FUNCTION_BLOCK PIDBase (* Composite Function Block Type *)
  (* Standard: 61499-2 *)
  (* Version 1.0.1, 10/18/2023, ApplicationLibDevTeam, Schneider Electric, First Version *)
  PACKAGE Main;
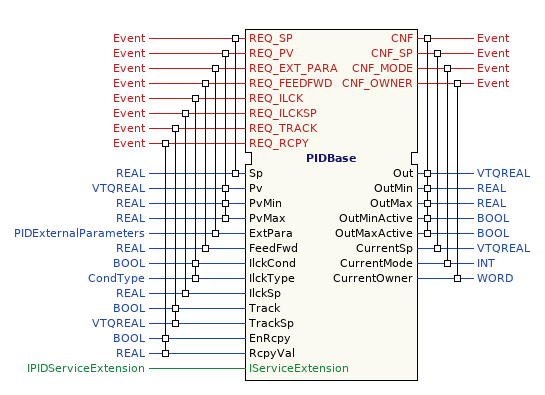
  EVENT_INPUT
    REQ_SP WITH Sp; (* Request to update setpoint *)
    REQ_PV WITH Pv, PvMin, PvMax; (* Request to update input value *)
    REQ_EXT_PARA WITH ExtPara; (* Request to update external PID parameters *)
    REQ_FEEDFWD WITH FeedFwd; (* Request for executing feed forward gain *)
    REQ_ILCK WITH IlckCond, IlckType; (* Request to update interlock conditions *)
    REQ_ILCKSP WITH IlckSp; (* Request to update interlock setpoint to PID ouput *)
    REQ_TRACK WITH Track, TrackSp; (* Request to track PID setpoint with TrackState *)
    REQ_RCPY WITH EnRcpy, RcpyVal; (* Request for actuator position *)
  END_EVENT
  EVENT_OUTPUT
    CNF WITH Out, OutMinActive, OutMaxActive, OutMin, OutMax; (* Execution confirmation (Cyclic update) *)
    CNF_SP WITH CurrentSp; (* Execution confirmation of current setpoint *)
    CNF_MODE WITH CurrentMode; (* Execution of confirmation of current mode *)
    CNF_OWNER WITH CurrentOwner; (* Execution confirmation of owner *)
  END_EVENT
  VAR_INPUT
    Sp : REAL; (* Setpoint for PID calculation *)
    Pv : VTQREAL; (* Unscaled analog process value *)
    PvMin : REAL; (* Minimum range of process value *)
    PvMax : REAL; (* Maximum range of process value *)
    ExtPara : PIDExternalParameters; (* External parameters for PID calculation *)
    FeedFwd : REAL; (* Feed forward value *)
    IlckCond : BOOL; (* 1 = Interlock condition active *)
    IlckType : CondType; (* Type of condition interlock, (0 = Normal, 1 = Process interlock/Sequence interlock) *)
    IlckSp : REAL; (* Interlock setpoint *)
    Track : BOOL; (* 1 = Track calclated output to TrackSp *)
    TrackSp : VTQREAL; (* If Track enabled, PID ouput follows TrackSp (Out = TrackSp) *)
    EnRcpy : BOOL; (* 1 = the RCPY is enabled *)
    RcpyVal : REAL; (* RCPY value (actuator position) *)
  END_VAR
  VAR_OUTPUT
    Out : VTQREAL; (* Calculated output value *)
    OutMin : REAL; (* Minimum range of ouput value *)
    OutMax : REAL; (* Maximum range of ouput value *)
    OutMinActive : BOOL; (* 1 = Out has reached OutMin Limit *)
    OutMaxActive : BOOL; (* 1 = Out has reached OutMax Limit *)
    CurrentSp : VTQREAL; (* Current setpoint value *)
    CurrentMode : INT; (* Current mode selected for PID calculation *)
    CurrentOwner : WORD; (* Current owner data from externlal source and basic owner 16#8 = Program owner, 16#10 = Operator owner, 16#4 = program Local and 16#40 Operator Local *)
  END_VAR
  SOCKETS
    IServiceExtension : IPIDServiceExtension(ServiceState := TRUE); (* Services extension adapter(Seq control and Owner) *)
  END_SOCKETS
  (* Initialization *)
  (* Supervision Interface *)
  (* Control *)
  (* Owner & Setpoint Management *)
  (* Data exchange with sequence *)
  (* Parameter Selection *)
  FBS
    IThis : PIDBase_HMI(QI := TRUE);
    plcStart : plcStart(Delay := T#0ms, Prio := 16);
    setpointRamp : rampCtl(MaxDeviation := 0.0, EnableDeviation := FALSE);
    pidCalc : pidCtl(ProhibitOutInc := FALSE, ProhibitOutDec := FALSE);
    modeSelection : devInSel(EnBumpless1 := FALSE, Val1 := (value:=0,quality:=16#0,timestamp:=LDT#2023-10-14-17:35:08,picosecs:=0), EnBumpless2 := TRUE, EnBumpless3 := FALSE, PermPassive := FALSE, PermActive1 := FALSE, PermActive2 := FALSE, UseCurrentVal := TRUE); {SET_ATTRIBUTE(Configuration.Component.HideUnusedPorts, )}
    basicOwner : ownerControl;
    programModeSelection : SELECT_24363B89CFDE21263(IN1 := 1); {SET_ATTRIBUTE(Configuration.GenericFBType.InterfaceParams, Runtime.Standard#CNT:=2;SELECT:BOOL;IN${CNT$}:INT)}
    spSelection : devRealSel(EnBumpless2 := TRUE, EnBumpless3 := FALSE, EnBumpless1 := FALSE); {SET_ATTRIBUTE(Configuration.Component.HideUnusedPorts, )}
    programSpSelection : SELECT_218F0E76F8A148ECD; {SET_ATTRIBUTE(Configuration.GenericFBType.InterfaceParams, Runtime.Standard#CNT:=2;SELECT:BOOL;IN${CNT$}:REAL)}
    outSelection : devRealSel(EnBumpless2 := FALSE, EnBumpless3 := TRUE, EnBumpless1 := FALSE, EnBumpless4 := FALSE, EnBumpless5 := FALSE); {SET_ATTRIBUTE(Configuration.Component.HideUnusedPorts, )}
    modeCalc : modeCalc;
    trackingActive : E_SELECT;
    paraSel : DS_SELECTX_125F0E43806CD1F46; {SET_ATTRIBUTE(Configuration.GenericFBType.InterfaceParams, Runtime.Standard#CNTX:=2;CNTY:=9;DI${CNTX,_,CNTY$}:REAL,REAL,REAL,BOOL,REAL,BOOL,REAL,REAL,REAL)} {SET_ATTRIBUTE(Configuration.Component.HideUnusedPorts, )}
    extParaSel : E_SWITCH;
    paraSelectionCheck : DS_SELECTX_4480AAC7B40EACCE; {SET_ATTRIBUTE(Configuration.GenericFBType.InterfaceParams, Runtime.Standard#CNTX:=2;CNTY:=10;DI${CNTX,_,CNTY$}:BOOL,REAL,REAL,REAL,BOOL,REAL,BOOL,REAL,REAL,REAL)}
    extParaCheck : E_SWITCH;
    paraSplit : SPLIT_62F891E498C2EEC3; {SET_ATTRIBUTE(Configuration.GenericFBType.InterfaceParams, Runtime.Standard#<InterfaceList> <EventInputs> <Event Name="REQ" Comment="Request events for dedicated input data sets"> <With Var="Input" /> </Event> </EventInputs> <EventOutputs> <Event Name="CNF" Comment="Confirmation from Resource for a dedicated request"> <With Var="Output" /> <With Var="Enable" /> <With Var="Gain" /> <With Var="IntegralTime" /> <With Var="DerivationTime" /> <With Var="Directon" /> <With Var="DeadBand" /> <With Var="DWorkOnError" /> <With Var="LagTime" /> <With Var="OutMin" /> <With Var="OutMax" /> </Event> </EventOutputs> <InputVars> <VarDeclaration Name="Input" Type="PIDExternalParameters" Namespace="SE.App2CommonProcess" /> </InputVars> <OutputVars> <VarDeclaration Name="Output" Type="PIDExternalParameters" Namespace="SE.App2CommonProcess" /> <VarDeclaration Name="Enable" Type="BOOL" /> <VarDeclaration Name="Gain" Type="REAL" /> <VarDeclaration Name="IntegralTime" Type="REAL" /> <VarDeclaration Name="DerivationTime" Type="REAL" /> <VarDeclaration Name="Directon" Type="BOOL" /> <VarDeclaration Name="DeadBand" Type="REAL" /> <VarDeclaration Name="DWorkOnError" Type="BOOL" /> <VarDeclaration Name="LagTime" Type="REAL" /> <VarDeclaration Name="OutMin" Type="REAL" /> <VarDeclaration Name="OutMax" Type="REAL" /> </OutputVars> </InterfaceList>)}
  END_FBS
  EVENT_CONNECTIONS
    modeSelection.CNF TO CNF_MODE;
    programSpSelection.CNF TO spSelection.REQ_SP3;
    programModeSelection.CNF TO modeSelection.REQ_SP3;
    IServiceExtension.REQ_OWNER TO basicOwner.REQ_STDOWNER;
    spSelection.CNF TO CNF_SP;
    REQ_TRACK TO modeSelection.REQ_SP1;
    REQ_ILCK TO outSelection.REQ_SEL;
    REQ_TRACK TO modeCalc.REQ_TRACK;
    REQ_TRACK TO outSelection.REQ_SP1;
    modeCalc.CNF TO outSelection.REQ_SEL;
    modeCalc.CNF_TRACK TO outSelection.REQ_SEL;
    REQ_ILCKSP TO outSelection.REQ_SP2;
    pidCalc.C_CNF TO outSelection.REQ_SP5;
    outSelection.CNF TO pidCalc.REQ;
    modeSelection.CNF TO modeCalc.REQ_MODE;
    modeCalc.CNF_TRACK TO modeSelection.REQ_SEL;
    IServiceExtension.REQ_CMD TO programModeSelection.REQ;
    IServiceExtension.REQ_SP TO programSpSelection.REQ;
    REQ_SP TO programSpSelection.REQ;
    REQ_PV TO pidCalc.REQ;
    modeCalc.CNF TO spSelection.REQ_SEL;
    REQ_PV TO spSelection.REQ_SP1;
    modeCalc.CNF TO setpointRamp.REQ_TRACK;
    spSelection.CNF TO setpointRamp.REQ_SP;
    modeSelection.CNF TO IServiceExtension.CNF_MODE;
    REQ_PV TO setpointRamp.REQ_SP;
    setpointRamp.CNF TO pidCalc.REQ_SP;
    REQ_FEEDFWD TO pidCalc.REQ_FEEDFWD;
    modeCalc.CNF_MODE TO pidCalc.REQ;
    REQ_PV TO setpointRamp.REQ_TRACK;
    REQ_ILCK TO IServiceExtension.CNF_READY;
    REQ_PV TO IServiceExtension.CNF_PV;
    setpointRamp.CNF TO IServiceExtension.CNF_SP_OP;
    plcStart.FIRST_INIT TO IServiceExtension.CNF_SERVICE;
    pidCalc.CNF_READY TO IServiceExtension.CNF_READY;
    basicOwner.CNF_OWNER TO modeCalc.REQ_OWNER;
    pidCalc.C_CNF TO trackingActive.EI0;
    trackingActive.EO TO CNF;
    modeCalc.CNF_TRACK TO trackingActive.EI0;
    trackingActive.EO TO IServiceExtension.CNF_SP_OP;
    pidCalc.CNF TO trackingActive.EI1;
    extParaSel.EO1 TO paraSel.REQ2;
    paraSel.IND TO pidCalc.REQ_PARA;
    REQ_TRACK TO pidCalc.REQ_TRACK;
    IServiceExtension.REQ_PARA TO extParaCheck.EI;
    extParaCheck.EO0 TO paraSelectionCheck.REQ1;
    extParaCheck.EO1 TO paraSelectionCheck.REQ2;
    REQ_EXT_PARA TO paraSplit.REQ;
    paraSplit.CNF TO extParaCheck.EI;
    IServiceExtension.REQ_OUT TO outSelection.REQ_SP4;
    REQ_ILCK TO modeCalc.REQ_ILCK;
    basicOwner.CNF_OWNER TO programModeSelection.REQ;
    REQ_TRACK TO IServiceExtension.CNF_TRACK;
    REQ_ILCK TO pidCalc.REQ_ILCK;
    modeCalc.CNF TO modeSelection.REQ_SEL;
    basicOwner.CNF_OWNER TO CNF_OWNER;
    paraSel.IND TO IServiceExtension.CNF_SP_OP;
    paraSel.IND TO IServiceExtension.8CDB19EE4FC593B1;
    paraSelectionCheck.IND TO extParaSel.EI;
    plcStart.FIRST_INIT TO IThis.F4ED48CC2B5317F8;
    IThis.3C7816C1E3C12126 TO IThis.F8BDFB66D6A721B;
    modeCalc.CNF TO IThis.4ECF71528D4B6340;
    REQ_ILCK TO IThis.4ECF71528D4B6340;
    REQ_PV TO IThis.4ECF71528D4B6340;
    setpointRamp.CNF TO IThis.4ECF71528D4B6340;
    pidCalc.CNF TO IThis.4ECF71528D4B6340;
    modeCalc.CNF_MODE TO IThis.4ECF71528D4B6340;
    REQ_TRACK TO IThis.4ECF71528D4B6340;
    pidCalc.C_CNF TO IThis.4ECF71528D4B6340;
    spSelection.CNF TO IThis.4ECF71528D4B6340;
    modeCalc.CNF_TRACK TO IThis.568B5274285BDEC8;
    paraSel.IND TO IThis.568B5274285BDEC8;
    extParaSel.EO0 TO IThis.568B5274285BDEC8;
    IThis.3C7816C1E3C12126 TO basicOwner.REQ_BASICOWNER;
    IThis.3C7816C1E3C12126 TO plcStart.ACK_FIRST;
    IThis.CF580EC7DC4C111C TO basicOwner.REQ_BASICOWNER;
    IThis.733DF8FD825824CA TO spSelection.REQ_SP2;
    IThis.F7A34A5B968DDB98 TO outSelection.REQ_SP3;
    IThis.DF1716734AF61076 TO setpointRamp.REQ_PARA;
    IThis.DF1716734AF61076 TO modeCalc.REQ_OWNER;
    IThis.DF1716734AF61076 TO paraSel.REQ1;
    IThis.D88CEB590B668985 TO modeSelection.REQ_SP2;
    IThis.D88CEB590B668985 TO setpointRamp.REQ_PARA;
    IThis.D88CEB590B668985 TO paraSel.REQ1;
    IThis.D716EC33D901A5A4 TO pidCalc.REQ_OUTBIAS;
    REQ_RCPY TO pidCalc.F3BAF1D546068DF6;
  END_CONNECTIONS
  DATA_CONNECTIONS
    modeSelection.CurrentVal TO CurrentMode;
    Sp TO programSpSelection.IN1;
    programSpSelection.OUT TO spSelection.Val3;
    programModeSelection.OUT TO modeSelection.Val3;
    basicOwner.ProgramOwner TO modeSelection.Sel3;
    basicOwner.OperatorOwner TO modeSelection.Sel2;
    basicOwner.StdOwnerConnected TO programModeSelection.SELECT;
    basicOwner.ProgramOwner TO spSelection.Sel3;
    basicOwner.StdOwnerConnected TO programSpSelection.SELECT;
    IServiceExtension.StdOwner TO basicOwner.StdOwner;
    spSelection.CurrentVal TO CurrentSp;
    TrackSp TO outSelection.Val1;
    Track TO modeSelection.Sel1;
    IlckSp TO outSelection.Val2;
    IlckCond TO outSelection.Sel2;
    Track TO outSelection.Sel1;
    Track TO modeCalc.Track;
    modeSelection.CurrentVal TO modeCalc.ModeIn;
    pidCalc.Out TO outSelection.Val5;
    outSelection.CurrentVal TO pidCalc.PresetValue;
    modeCalc.ModeOut TO outSelection.Sel5;
    modeCalc.OperManual TO outSelection.Sel3;
    IServiceExtension.Sp TO programModeSelection.IN2;
    IServiceExtension.SpReal1 TO programSpSelection.IN2;
    modeCalc.TrackManual TO spSelection.Sel1;
    Pv TO pidCalc.Pv;
    Pv TO spSelection.Val1;
    modeCalc.TrackManual TO setpointRamp.Track;
    IlckCond TO modeCalc.IlckCond;
    spSelection.CurrentVal TO setpointRamp.Sp;
    modeSelection.CurrentVal TO IServiceExtension.CurrentMode;
    PvMin TO setpointRamp.SpMin;
    PvMax TO setpointRamp.SpMax;
    Pv TO setpointRamp.TrackSp;
    setpointRamp.Out TO pidCalc.Sp;
    FeedFwd TO pidCalc.FeedFwd;
    IlckCond TO IServiceExtension.Interlocked;
    pidCalc.Out TO IServiceExtension.CurrentOp;
    setpointRamp.Out TO IServiceExtension.CurrentSp;
    Pv TO IServiceExtension.Pv;
    pidCalc.Out TO Out;
    pidCalc.OutMinActive TO OutMinActive;
    pidCalc.OutMaxActive TO OutMaxActive;
    IlckType TO pidCalc.IlckType;
    IlckCond TO pidCalc.IlckCond;
    pidCalc.Ready TO IServiceExtension.Ready;
    Track TO pidCalc.TrackSp;
    modeCalc.OperAuto TO spSelection.Sel2;
    basicOwner.Owner TO modeCalc.Owner;
    Track TO trackingActive.G;
    modeCalc.ProgLocalManual TO outSelection.Sel4;
    paraSel.OUT1 TO pidCalc.Gain;
    paraSel.OUT2 TO pidCalc.IntegralTime;
    paraSel.OUT3 TO pidCalc.DerivativeTime;
    paraSel.OUT4 TO pidCalc.Direction;
    paraSel.OUT5 TO pidCalc.Deadband;
    paraSel.OUT6 TO pidCalc.DWorkOnError;
    paraSel.OUT7 TO pidCalc.LagTime;
    paraSel.OUT8 TO pidCalc.OutMin;
    paraSel.OUT9 TO pidCalc.OutMax;
    IServiceExtension.ExtParaSel TO extParaCheck.G;
    IServiceExtension.Gain TO paraSelectionCheck.DI2_2;
    IServiceExtension.IntegralTime TO paraSelectionCheck.DI2_3;
    IServiceExtension.DerivationTime TO paraSelectionCheck.DI2_4;
    IServiceExtension.Direction TO paraSelectionCheck.DI2_5;
    IServiceExtension.DeadBand TO paraSelectionCheck.DI2_6;
    IServiceExtension.DWorkOnError TO paraSelectionCheck.DI2_7;
    IServiceExtension.LagTime TO paraSelectionCheck.DI2_8;
    IServiceExtension.OutMin TO paraSelectionCheck.DI2_9;
    IServiceExtension.OutMax TO paraSelectionCheck.DI2_10;
    paraSel.OUT8 TO OutMin;
    paraSel.OUT9 TO OutMax;
    paraSelectionCheck.OUT10 TO paraSel.DI2_9;
    paraSelectionCheck.OUT2 TO paraSel.DI2_1;
    paraSelectionCheck.OUT3 TO paraSel.DI2_2;
    paraSelectionCheck.OUT4 TO paraSel.DI2_3;
    paraSelectionCheck.OUT5 TO paraSel.DI2_4;
    paraSelectionCheck.OUT6 TO paraSel.DI2_5;
    paraSelectionCheck.OUT7 TO paraSel.DI2_6;
    paraSelectionCheck.OUT8 TO paraSel.DI2_7;
    paraSelectionCheck.OUT9 TO paraSel.DI2_8;
    IServiceExtension.ExtParaSel TO paraSelectionCheck.DI2_1;
    paraSelectionCheck.OUT1 TO extParaSel.G;
    ExtPara TO paraSplit.Input;
    paraSplit.Enable TO paraSelectionCheck.DI1_1;
    paraSplit.Gain TO paraSelectionCheck.DI1_2;
    paraSplit.IntegralTime TO paraSelectionCheck.DI1_3;
    paraSplit.DerivationTime TO paraSelectionCheck.DI1_4;
    paraSplit.Directon TO paraSelectionCheck.DI1_5;
    paraSplit.DeadBand TO paraSelectionCheck.DI1_6;
    paraSplit.DWorkOnError TO paraSelectionCheck.DI1_7;
    paraSplit.LagTime TO paraSelectionCheck.DI1_8;
    paraSplit.OutMin TO paraSelectionCheck.DI1_9;
    paraSplit.OutMax TO paraSelectionCheck.DI1_10;
    IServiceExtension.SpReal2 TO outSelection.Val4;
    modeCalc.CalcMode TO pidCalc.Mode;
    Track TO IServiceExtension.Track;
    basicOwner.Owner TO CurrentOwner;
    PvMin TO IServiceExtension.PvMin;
    PvMax TO IServiceExtension.PvMax;
    paraSel.OUT8 TO IServiceExtension.CurrentOpMin;
    paraSel.OUT9 TO IServiceExtension.CurrentOpMax;
    paraSel.OUT1 TO IServiceExtension.526988CF984C619A;
    paraSel.OUT2 TO IServiceExtension.7D8F5388E2DC486D;
    paraSel.OUT3 TO IServiceExtension.B62ECEA2F5E6DA8A;
    paraSel.OUT4 TO IServiceExtension.607F2E8B0E693249;
    paraSel.OUT5 TO IServiceExtension.60EB9615BA837102;
    paraSel.OUT6 TO IServiceExtension.3F4910500F1CC6A6;
    paraSel.OUT7 TO IServiceExtension.B38B3033E4F94F3F;
    Pv TO IThis.ACDC6904590859A8;
    PvMin TO IThis.8881FFD24D90D865;
    PvMax TO IThis.E15A9214DEEE85B6;
    spSelection.CurrentVal TO IThis.AA9BE811C6AB052A;
    pidCalc.Out TO IThis.F680A73B417CD6F5;
    modeSelection.CurrentVal TO IThis.5BB4B57D9CC10C19;
    basicOwner.Owner TO IThis.3143D32BCC6D529B;
    pidCalc.OutChangeProhibited TO IThis.38051CE7590A4498;
    Track TO IThis.F23EE025A922C157;
    pidCalc.Outbias TO IThis.A375666527EF676C;
    IlckCond TO IThis.2F039F336E3FD06B;
    paraSelectionCheck.OUT1 TO IThis.B2A8B3D1DEEA17E;
    paraSel.OUT1 TO IThis.9687AF2C021C1405;
    paraSel.OUT2 TO IThis.34E69DFE80FEB19D;
    paraSel.OUT3 TO IThis.DF0E3B1C6754334E;
    paraSel.OUT4 TO IThis.D797C0265258257A;
    paraSel.OUT5 TO IThis.2D62610692B0BAA7;
    paraSel.OUT6 TO IThis.59BC22F58A2AC5DE;
    paraSel.OUT7 TO IThis.DFD108CBF0371C9F;
    paraSel.OUT8 TO IThis.6582E689B1B84E24;
    paraSel.OUT9 TO IThis.43713152FBB271A0;
    basicOwner.StdOwnerConnected TO IThis.659F42A0E6591C81;
    IThis.45D13D51972F673D TO basicOwner.BasicOwner;
    IThis.85E36F6C7A7A3394 TO spSelection.Val2;
    IThis.99DCC6ECF79655A0 TO outSelection.Val3;
    IThis.8B3FE585BEF5C081 TO modeSelection.Val2;
    IThis.91FE3D159818E304 TO paraSel.DI1_1;
    IThis.7A7AC172CDE65711 TO paraSel.DI1_2;
    IThis.885D832E4B845B40 TO paraSel.DI1_3;
    IThis.5A6B0DD7FD7B5424 TO paraSel.DI1_4;
    IThis.BB44C6E631F7BD3C TO paraSel.DI1_5;
    IThis.6FC912D3B6844A9C TO paraSel.DI1_6;
    IThis.802873E984BC2734 TO paraSel.DI1_7;
    IThis.40822142BE6CD80A TO paraSel.DI1_8;
    IThis.E96A0C6730BB0132 TO paraSel.DI1_9;
    IThis.5A03B435FD6E1D89 TO setpointRamp.CycleTime;
    IThis.5A03B435FD6E1D89 TO pidCalc.CycleTime;
    IThis.598D23039F0AFA46 TO pidCalc.EnFeedFwd;
    IThis.5C7C217636F1BA76 TO pidCalc.FeedFwdGain;
    IThis.5CE0359990D76374 TO pidCalc.Bump;
    IThis.B2E2120DF5C5B08 TO pidCalc.OutbiasOffset;
    IThis.F5B64A07FB2C2078 TO setpointRamp.RateUp;
    IThis.2AF043299B6A959D TO setpointRamp.RateDown;
    IThis.4568BE33B21F361B TO modeCalc.EnManualTrackSp;
    IThis.2674CCA549C60F52 TO pidCalc.92AFF823C3B58F8C;
    IThis.F385201F0CB7361F TO pidCalc.7B1B4A8898E5166E;
    IThis.896A9B3CA40C38E3 TO pidCalc.1D9F3DDE91AAFB44;
    EnRcpy TO pidCalc.26A58A49358F5359;
    RcpyVal TO pidCalc.EB9D275C1F9B5CB3;
  END_CONNECTIONS
END_FUNCTION_BLOCK
